{attribute 'qualified_only'}
VAR_GLOBAL
  Com : ZCom;
END_VAR
VAR_GLOBAL PERSISTENT
  Data : ZData;
END_VAR

(* stored: Version 1.1.0.1
   GVL ZGlobal: Id {922707fe-d804-424c-8a1a-a278bfaf408a} *)
